# EPICS autosave request: iocBoot/iocTXMOptics/auto_settings.req
file "txmOptics.req", P=$(P), R=$(R)
file "txmOptics_settings.req", P=$(P), R=$(R)
